SUBAPPLICATION Outputs (* Subapplication Type *)
  (* Standard: 61499-2 *)
  (* Version 1.0, 2025-01-31, franz *)
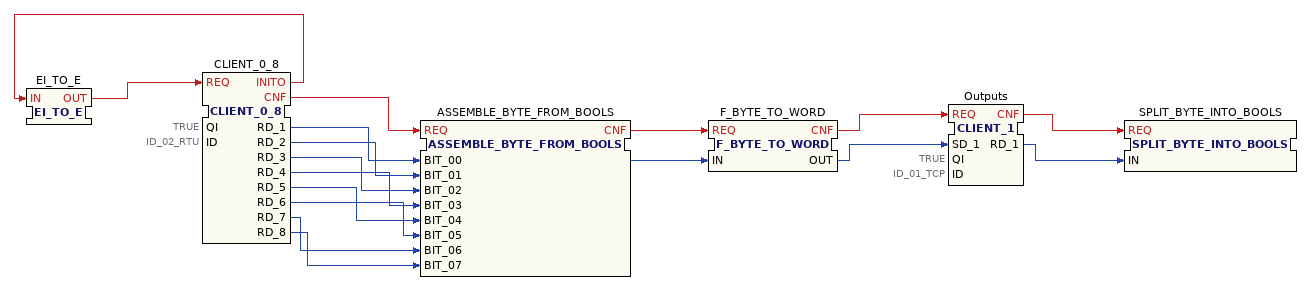
  FBS
    F_BYTE_TO_WORD : F_BYTE_TO_WORD;
    ASSEMBLE_BYTE_FROM_BOOLS : ASSEMBLE_BYTE_FROM_BOOLS;
    Outputs : CLIENT_1(QI := TRUE, ID := ID_01_TCP);
    SPLIT_BYTE_INTO_BOOLS : SPLIT_BYTE_INTO_BOOLS;
    CLIENT_0_8 : CLIENT_0_8(QI := TRUE, ID := ID_02_RTU);
    EI_TO_E : EI_TO_E;
  END_FBS
  EVENT_CONNECTIONS
    ASSEMBLE_BYTE_FROM_BOOLS.CNF TO F_BYTE_TO_WORD.REQ;
    F_BYTE_TO_WORD.CNF TO Outputs.REQ;
    Outputs.CNF TO SPLIT_BYTE_INTO_BOOLS.REQ;
    EI_TO_E.OUT TO CLIENT_0_8.REQ;
    CLIENT_0_8.INITO TO EI_TO_E.IN;
    CLIENT_0_8.CNF TO ASSEMBLE_BYTE_FROM_BOOLS.REQ;
  END_CONNECTIONS
  DATA_CONNECTIONS
    ASSEMBLE_BYTE_FROM_BOOLS. TO F_BYTE_TO_WORD.IN;
    F_BYTE_TO_WORD.OUT TO Outputs.SD_1;
    Outputs.RD_1 TO SPLIT_BYTE_INTO_BOOLS.IN;
    CLIENT_0_8.RD_1 TO ASSEMBLE_BYTE_FROM_BOOLS.BIT_00;
    CLIENT_0_8.RD_2 TO ASSEMBLE_BYTE_FROM_BOOLS.BIT_01;
    CLIENT_0_8.RD_3 TO ASSEMBLE_BYTE_FROM_BOOLS.BIT_02;
    CLIENT_0_8.RD_4 TO ASSEMBLE_BYTE_FROM_BOOLS.BIT_03;
    CLIENT_0_8.RD_5 TO ASSEMBLE_BYTE_FROM_BOOLS.BIT_04;
    CLIENT_0_8.RD_6 TO ASSEMBLE_BYTE_FROM_BOOLS.BIT_05;
    CLIENT_0_8.RD_7 TO ASSEMBLE_BYTE_FROM_BOOLS.BIT_06;
    CLIENT_0_8.RD_8 TO ASSEMBLE_BYTE_FROM_BOOLS.BIT_07;
  END_CONNECTIONS
END_SUBAPPLICATION
